FUNCTION_BLOCK Heating_State_Disabled EXTENDS Heating_State
VAR_INPUT
END_VAR
VAR_OUTPUT
END_VAR
VAR
END_VAR

METHOD OnInit
_ctx.hmi.sStatusText := 'Heating disabled!';
_ctx.hmi.nStatusColor := COL.BLACK.Raw;

_ctx.hmi.sButtonText := 'Press to ENABLE!';
_ctx.hmi.nButtonColor := COL.BLACK.Raw;

_ctx.io.out.bBurner := FALSE;
_ctx.io.out.bPump := FALSE;
END_METHOD

END_FUNCTION_BLOCK

(* stored: Version 1.1.0.1
   POU Heating_State_Disabled: Id {3b811875-1208-4731-9501-ae0d4edb08e7}, SpecialFunc None
   Method OnInit: Id {969084cd-eabe-4f07-bb36-9264c638a3be} *)
